{attribute 'qualified_only'}
VAR_GLOBAL
	
	//for reading as
	//dynamic gTOASTHMI = symbols["gTOASTHHMI"];
	gData:structHMIGlobal;
	
END_VAR

(* stored: Version 1.1.0.1, ProductVersion 3.1.4024.11
   GVL gTOASTHMI: Id {22590b88-a8ac-0347-0ff6-b6fe3895de21} *)
